VAR_GLOBAL
	MoverInfo: ARRAY[1..GrpCnt] OF DUT_MoverInfo;
	AwaitingReservationAxis: INT := 0;
	AwaitingAxisCnt: INT := 0;
	SkillAx:	ARRAY [1..GrpCnt] OF INT;
	Reservingaxis	: INT := 0;
	
END_VAR

(* stored: Version 1.1.0.1, ProductVersion 3.1.0.25
   GVL Mover_Infos: Id {186aac3b-ccb6-4fca-829d-336dddd1fac9} *)
